(* Logix 5000 project; controller GEA_Test_Chamber vendor 1 type 14 code 196 rev 32.14; software revision 32.04; part 5 of 11 *)
(* tags used below, declared in another part *)
   Wrk_Index : DINT;
(* raC_Tec_NetModbusTCPServer_RespStrWord, continued *)

ROUTINE Prescan   (* ladder *)
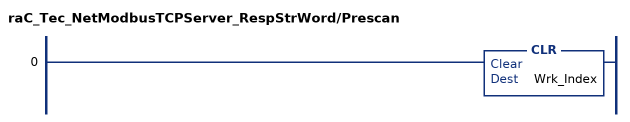
   0: CLR(Wrk_Index);
END_ROUTINE
END_ADD_ON_INSTRUCTION

ADD_ON_INSTRUCTION T_DIFF   (* revision 1.0 *)
VAR_IN_OUT
   TimeRef : DINT[7]; {required}
   ActTime : DINT[7]; {required}
END_VAR
VAR_OUTPUT
   T_Diff_sec : DINT; {required}
END_VAR
VAR
   Temp_Time : DINT[7]; {access None}
   sec : DINT[3]; {access None}
END_VAR

ROUTINE Logic   (* ladder *)
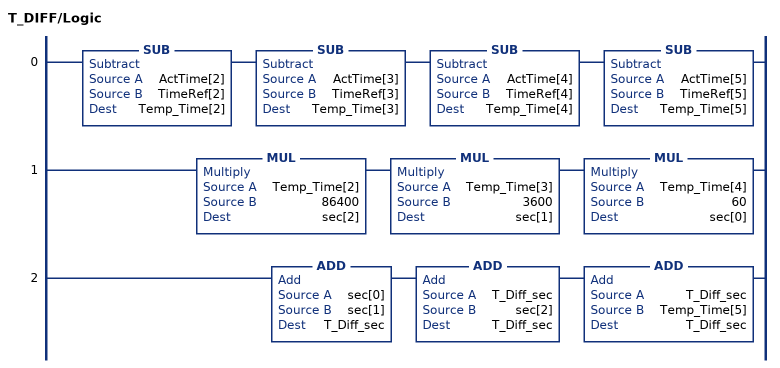
   0: SUB(ActTime[2],TimeRef[2],Temp_Time[2])SUB(ActTime[3],TimeRef[3],Temp_Time[3])SUB(ActTime[4],TimeRef[4],Temp_Time[4])SUB(ActTime[5],TimeRef[5],Temp_Time[5]);
   1: MUL(Temp_Time[2],86400,sec[2])MUL(Temp_Time[3],3600,sec[1])MUL(Temp_Time[4],60,sec[0]);
   2: ADD(sec[0],sec[1],T_Diff_sec)ADD(T_Diff_sec,sec[2],T_Diff_sec)ADD(T_Diff_sec,Temp_Time[5],T_Diff_sec);
END_ROUTINE
END_ADD_ON_INSTRUCTION

VAR_GLOBAL   (* controller tags *)
   always_off : BOOL;
   Amount_Water_Flow : DINT := 200;
   Client_01 : raC_Opr_NetModbusTCPClient := (Inp_Enable := 1, Sts_EN := 1, Sts_Connected := 1);
   Client_01_Data : raC_UDT_ModbusClientData := (Coils_0xxx[0] := 1, Coils_0xxx[1] := 1, Coils_0xxx[2] := 1, Coils_0xxx[3] := 1, Coils_0xxx[1010] := 1, Coils_0xxx[1012] := 1, Coils_0xxx[1014] := 1, Coils_0xxx[1015] := 1, HoldRegisters_4xxx[0] := 10, HoldRegisters_4xxx[1] := 512, HoldRegisters_4xxx[32] := 102, HoldRegisters_4xxx[33] := 2330);
   Client_01_EN : BOOL := 1;
   Client_01_MSG_Connect : MESSAGE;
        MessageParameters(ServiceCode := 16#004c, LocalElement := Client_01_Parameters.MSG_Src[0], ...)
   Client_01_MSG_Create : MESSAGE;
        MessageParameters(ServiceCode := 16#004b, LocalElement := Client_01_Parameters.MSG_Src[0], DestinationTag := Client_01_Parameters.MSG_Dest[0], ...)
   Client_01_MSG_Delete : MESSAGE;
        MessageParameters(ServiceCode := 16#004f, ...)
   Client_01_MSG_Read : MESSAGE;
        MessageParameters(ServiceCode := 16#004d, LocalElement := Client_01_Parameters.MSG_Src[0], DestinationTag := Client_01_Parameters.MSG_Dest[0], ...)
   Client_01_MSG_SetSing : MESSAGE;
        MessageParameters(ServiceCode := 16#0010, LocalElement := Client_01_Parameters.MSG_Src[496], ...)
   Client_01_MSG_Write : MESSAGE;
        MessageParameters(ServiceCode := 16#004e, LocalElement := Client_01_Parameters.MSG_Src[0], DestinationTag := Client_01_Parameters.MSG_Dest[0], ...)
   Client_01_Parameters : raC_UDT_ModbusClientConnection := (DestAddress := '10.2.0.15', DestinationPort := 502, MSG_Src[4] := -28, MSG_Src[5] := 1, MSG_Src[12] := 12, MSG_Src[16] := 58, MSG_Src[17] := 106, MSG_Src[21] := 6, MSG_Src[22] := 1, MSG_Src[23] := 4, MSG_Src[25] := 3, MSG_Src[27] := 10, MSG_Src[28] := 50, MSG_Src[29] := 50, MSG_Src[496] := 1, MSG_Dest[12] := 58, MSG_Dest[13] := 105, MSG_Dest[17] := 23, MSG_Dest[18] := 1, MSG_Dest[19] := 4, MSG_Dest[20] := 20, MSG_Dest[86] := 102, MSG_Dest[87] := 9, MSG_Dest[88] := 26, MSG_Dest[232] := 105, MSG_Dest[233] := 29, MSG_Dest[237] := 6, MSG_Dest[239] := 6);
   Client_01_Transactions : raC_UDT_ModbusClientTransaction[5] := ([0].Enabled := 1, [0].PollInterval := 500, [0].TransType := 4, [0].StationID := 1, [0].BeginAddress := 3, [0].Count := 10, [0].TransComplete := 1, [0].Diagnostic.Request := ':h$00$00$00$06$01$04$00$03$00$0A', [0].Diagnostic.TransID := 14952, [0].Diagnostic.IntervalTimer.PRE := 460, [0].Diagnostic.IntervalTimer.ACC := 395, [0].Diagnostic.IntervalTimer.EN := 1, [0].Diagnostic.IntervalTimer.TT := 1, [0].Diagnostic.NoReplyCounter.PRE := 10, [0].Diagnostic.PendingTimer.PRE := 3000, [1].PollInterval := 1000, [1].Diagnostic.IntervalTimer.PRE := 960, [1].Diagnostic.IntervalTimer.ACC := 960, [1].Diagnostic.IntervalTimer.EN := 1, [1].Diagnostic.IntervalTimer.DN := 1, [1].Diagnostic.NoReplyCounter.PRE := 10, [1].Diagnostic.PendingTimer.PRE := 3000, [2].PollInterval := 1000, [2].Diagnostic.IntervalTimer.PRE := 960, [2].Diagnostic.IntervalTimer.ACC := 960, [2].Diagnostic.IntervalTimer.EN := 1, [2].Diagnostic.IntervalTimer.DN := 1, [2].Diagnostic.NoReplyCounter.PRE := 10, [2].Diagnostic.PendingTimer.PRE := 3000, [3].PollInterval := 1000, [3].Diagnostic.IntervalTimer.PRE := 960, [3].Diagnostic.IntervalTimer.ACC := 960, [3].Diagnostic.IntervalTimer.EN := 1, [3].Diagnostic.IntervalTimer.DN := 1, [3].Diagnostic.NoReplyCounter.PRE := 10, [3].Diagnostic.PendingTimer.PRE := 3000, [4].PollInterval := 1000, [4].Diagnostic.IntervalTimer.PRE := 960, [4].Diagnostic.IntervalTimer.ACC := 369, [4].Diagnostic.IntervalTimer.EN := 1, [4].Diagnostic.IntervalTimer.DN := 1, [4].Diagnostic.NoReplyCounter.PRE := 10, [4].Diagnostic.PendingTimer.PRE := 3000);
   Client_02 : raC_Opr_NetModbusTCPClient := (Inp_Enable := 1, Sts_EN := 1, Sts_Connected := 1);
   Client_02_Data : raC_UDT_ModbusClientData := (Coils_0xxx[0] := 1, Coils_0xxx[1] := 1, Coils_0xxx[2] := 1, Coils_0xxx[3] := 1, Coils_0xxx[1010] := 1, Coils_0xxx[1012] := 1, Coils_0xxx[1014] := 1, Coils_0xxx[1015] := 1, InpRegisters_3xxx[3] := 159, InpRegisters_3xxx[7] := 1904);
   Client_02_EN : BOOL := 1;
   Client_02_MSG_Connect : MESSAGE;
        MessageParameters(ServiceCode := 16#004c, LocalElement := Client_02_Parameters.MSG_Src[0], ...)
   Client_02_MSG_Create : MESSAGE;
        MessageParameters(ServiceCode := 16#004b, LocalElement := Client_02_Parameters.MSG_Src[0], DestinationTag := Client_02_Parameters.MSG_Dest[0], ...)
   Client_02_MSG_Delete : MESSAGE;
        MessageParameters(ServiceCode := 16#004f, ...)
   Client_02_MSG_Read : MESSAGE;
        MessageParameters(ServiceCode := 16#004d, LocalElement := Client_02_Parameters.MSG_Src[0], DestinationTag := Client_02_Parameters.MSG_Dest[0], ...)
   Client_02_MSG_SetSing : MESSAGE;
        MessageParameters(ServiceCode := 16#0010, LocalElement := Client_02_Parameters.MSG_Src[496], ...)
   Client_02_MSG_Write : MESSAGE;
        MessageParameters(ServiceCode := 16#004e, LocalElement := Client_02_Parameters.MSG_Src[0], DestinationTag := Client_02_Parameters.MSG_Dest[0], ...)
   Client_02_Parameters : raC_UDT_ModbusClientConnection := (DestAddress := '10.2.0.14', DestinationPort := 502, MSG_Src[4] := -28, MSG_Src[5] := 1, MSG_Src[12] := 12, MSG_Src[16] := 63, MSG_Src[17] := 53, MSG_Src[21] := 6, MSG_Src[22] := 1, MSG_Src[23] := 4, MSG_Src[25] := 3, MSG_Src[27] := 10, MSG_Src[28] := 20, MSG_Src[496] := 1, MSG_Dest[12] := 63, MSG_Dest[13] := 52, MSG_Dest[17] := 23, MSG_Dest[18] := 1, MSG_Dest[19] := 4, MSG_Dest[20] := 20, MSG_Dest[28] := -97, MSG_Dest[35] := 7, MSG_Dest[36] := 112, MSG_Dest[42] := 1, MSG_Dest[43] := -122, MSG_Dest[44] := -96, MSG_Dest[45] := 48, MSG_Dest[46] := 50, MSG_Dest[47] := 48, MSG_Dest[48] := 46, MSG_Dest[49] := 51, MSG_Dest[50] := 52, MSG_Dest[51] := 32, MSG_Dest[52] := 48, MSG_Dest[53] := 48, MSG_Dest[54] := 50, MSG_Dest[55] := 48, MSG_Dest[56] := 46, MSG_Dest[57] := 51, MSG_Dest[58] := 52, MSG_Dest[59] := 32, MSG_Dest[60] := 48, MSG_Dest[61] := 48, MSG_Dest[62] := 50, MSG_Dest[63] := 48, MSG_Dest[64] := 46, MSG_Dest[65] := 51, MSG_Dest[66] := 52, MSG_Dest[67] := 32, MSG_Dest[68] := 48, MSG_Dest[69] := 48, MSG_Dest[70] := 50, MSG_Dest[71] := 48, MSG_Dest[72] := 46, MSG_Dest[73] := 51, MSG_Dest[74] := 52, MSG_Dest[75] := 32, MSG_Dest[76] := 48, MSG_Dest[77] := 48, MSG_Dest[78] := 50,
        MSG_Dest[79] := 48, MSG_Dest[80] := 46, MSG_Dest[81] := 51, MSG_Dest[82] := 52, MSG_Dest[83] := 32, MSG_Dest[84] := 48, MSG_Dest[85] := 48, MSG_Dest[86] := 50, MSG_Dest[87] := 48, MSG_Dest[88] := 46, MSG_Dest[89] := 51, MSG_Dest[90] := 52, MSG_Dest[91] := 32, MSG_Dest[92] := 48, MSG_Dest[93] := 48, MSG_Dest[94] := 50, MSG_Dest[95] := 48, MSG_Dest[96] := 46, MSG_Dest[97] := 51, MSG_Dest[98] := 52, MSG_Dest[99] := 32, MSG_Dest[100] := 48, MSG_Dest[101] := 48, MSG_Dest[102] := 50, MSG_Dest[103] := 48, MSG_Dest[104] := 46, MSG_Dest[105] := 51, MSG_Dest[106] := 52, MSG_Dest[107] := 32, MSG_Dest[108] := 48, MSG_Dest[109] := 48, MSG_Dest[110] := 50, MSG_Dest[111] := 48, MSG_Dest[112] := 46, MSG_Dest[113] := 51, MSG_Dest[114] := 52, MSG_Dest[115] := 32, MSG_Dest[116] := 48, MSG_Dest[117] := 48, MSG_Dest[118] := 50, MSG_Dest[119] := 48, MSG_Dest[120] := 46, MSG_Dest[121] := 51, MSG_Dest[122] := 52, MSG_Dest[123] := 32, MSG_Dest[124] := 48, MSG_Dest[125] := 48, MSG_Dest[126] := 50, MSG_Dest[127] := 48, MSG_Dest[128] := 46, MSG_Dest[129] := 51, MSG_Dest[130] := 52, MSG_Dest[131] := 32, MSG_Dest[132] := 48, MSG_Dest[133] := 48, MSG_Dest[134] := 50, MSG_Dest[135] := 48, MSG_Dest[136] := 46, MSG_Dest[137] := 51, MSG_Dest[138] := 52,
        MSG_Dest[139] := 32, MSG_Dest[140] := 48, MSG_Dest[141] := 48, MSG_Dest[142] := 50, MSG_Dest[143] := 48, MSG_Dest[144] := 46, MSG_Dest[145] := 51, MSG_Dest[146] := 52, MSG_Dest[147] := 32, MSG_Dest[148] := 48, MSG_Dest[149] := 48, MSG_Dest[150] := 50, MSG_Dest[151] := 48, MSG_Dest[152] := 46, MSG_Dest[153] := 51, MSG_Dest[154] := 52, MSG_Dest[155] := 32, MSG_Dest[156] := 48, MSG_Dest[157] := 48, MSG_Dest[158] := 50, MSG_Dest[159] := 48, MSG_Dest[160] := 46, MSG_Dest[161] := 51, MSG_Dest[162] := 52, MSG_Dest[163] := 32, MSG_Dest[164] := 48, MSG_Dest[165] := 48, MSG_Dest[166] := 50, MSG_Dest[167] := 48, MSG_Dest[168] := 46, MSG_Dest[169] := 51, MSG_Dest[170] := 52, MSG_Dest[171] := 32, MSG_Dest[172] := 48, MSG_Dest[173] := 48, MSG_Dest[174] := 50, MSG_Dest[175] := 48, MSG_Dest[176] := 46, MSG_Dest[177] := 51, MSG_Dest[178] := 52, MSG_Dest[179] := 32, MSG_Dest[180] := 48, MSG_Dest[181] := 48, MSG_Dest[182] := 50, MSG_Dest[183] := 48, MSG_Dest[184] := 46, MSG_Dest[185] := 51, MSG_Dest[186] := 52, MSG_Dest[187] := 32, MSG_Dest[188] := 48, MSG_Dest[189] := 48, MSG_Dest[190] := 50, MSG_Dest[191] := 48, MSG_Dest[192] := 46, MSG_Dest[193] := 51, MSG_Dest[194] := 52, MSG_Dest[195] := 32, MSG_Dest[196] := 48, MSG_Dest[197] := 48, MSG_Dest[198] := 50,
        MSG_Dest[199] := 48, MSG_Dest[200] := 46, MSG_Dest[201] := 51, MSG_Dest[202] := 52, MSG_Dest[203] := 32, MSG_Dest[204] := 48, MSG_Dest[205] := 48, MSG_Dest[206] := 50, MSG_Dest[207] := 48, MSG_Dest[208] := 46, MSG_Dest[209] := 51, MSG_Dest[210] := 52, MSG_Dest[211] := 32, MSG_Dest[212] := 48, MSG_Dest[213] := 48, MSG_Dest[214] := 50, MSG_Dest[215] := 48, MSG_Dest[216] := 46, MSG_Dest[217] := 51, MSG_Dest[218] := 52, MSG_Dest[219] := 32, MSG_Dest[220] := 48, MSG_Dest[221] := 48, MSG_Dest[222] := 50, MSG_Dest[223] := 48, MSG_Dest[224] := 46, MSG_Dest[225] := 51, MSG_Dest[226] := 52, MSG_Dest[227] := 32, MSG_Dest[228] := 48, MSG_Dest[229] := 48, MSG_Dest[230] := 50, MSG_Dest[231] := 48, MSG_Dest[232] := 46, MSG_Dest[233] := 51, MSG_Dest[234] := 52, MSG_Dest[235] := 32, MSG_Dest[236] := 48, MSG_Dest[237] := 48, MSG_Dest[238] := 50, MSG_Dest[239] := 48, MSG_Dest[240] := 46, MSG_Dest[241] := 51, MSG_Dest[242] := 52, MSG_Dest[243] := 32, MSG_Dest[244] := 48, MSG_Dest[245] := 48, MSG_Dest[246] := 50, MSG_Dest[247] := 48, MSG_Dest[248] := 46, MSG_Dest[249] := 51, MSG_Dest[250] := 52, MSG_Dest[251] := 32, MSG_Dest[252] := 48, MSG_Dest[253] := 48, MSG_Dest[254] := 50, MSG_Dest[255] := 48, MSG_Dest[256] := 46, MSG_Dest[257] := 51, MSG_Dest[258] := 52,
        MSG_Dest[259] := 32, MSG_Dest[260] := 48, MSG_Dest[261] := 48, MSG_Dest[262] := 50, MSG_Dest[263] := 48, MSG_Dest[264] := 46, MSG_Dest[265] := 51, MSG_Dest[266] := 52, MSG_Dest[267] := 32);
   Client_02_Transactions : raC_UDT_ModbusClientTransaction[5] := ([0].Enabled := 1, [0].PollInterval := 500, [0].TransType := 4, [0].StationID := 1, [0].BeginAddress := 3, [0].Count := 10, [0].TransStat := 1, [0].Diagnostic.Request := '?4$00$00$00$06$01$04$00$03$00$0A', [0].Diagnostic.ReqBuilt := 1, [0].Diagnostic.TransID := 16180, [0].Diagnostic.IntervalTimer.PRE := 460, [0].Diagnostic.IntervalTimer.ACC := 44, [0].Diagnostic.IntervalTimer.EN := 1, [0].Diagnostic.IntervalTimer.TT := 1, [0].Diagnostic.NoReplyCounter.PRE := 10, [0].Diagnostic.PendingTimer.PRE := 3000, [0].Diagnostic.PendingTimer.ACC := 44, [0].Diagnostic.PendingTimer.EN := 1, [0].Diagnostic.PendingTimer.TT := 1, [1].PollInterval := 1000, [1].Diagnostic.IntervalTimer.PRE := 960, [1].Diagnostic.IntervalTimer.ACC := 960, [1].Diagnostic.IntervalTimer.EN := 1, [1].Diagnostic.IntervalTimer.DN := 1, [1].Diagnostic.NoReplyCounter.PRE := 10, [1].Diagnostic.PendingTimer.PRE := 3000, [2].PollInterval := 1000, [2].Diagnostic.IntervalTimer.PRE := 960, [2].Diagnostic.IntervalTimer.ACC := 960, [2].Diagnostic.IntervalTimer.EN := 1, [2].Diagnostic.IntervalTimer.DN := 1, [2].Diagnostic.NoReplyCounter.PRE := 10, [2].Diagnostic.PendingTimer.PRE := 3000, [3].PollInterval := 1000, [3].Diagnostic.IntervalTimer.PRE := 960, [3].Diagnostic.IntervalTimer.ACC := 369, [3].Diagnostic.IntervalTimer.EN := 1, [3].Diagnostic.IntervalTimer.DN := 1, [3].Diagnostic.NoReplyCounter.PRE := 10, [3].Diagnostic.PendingTimer.PRE := 3000, [4].PollInterval := 1000, [4].Diagnostic.IntervalTimer.PRE := 960, [4].Diagnostic.IntervalTimer.ACC := 369, [4].Diagnostic.IntervalTimer.EN := 1, [4].Diagnostic.IntervalTimer.DN := 1, [4].Diagnostic.NoReplyCounter.PRE := 10, [4].Diagnostic.PendingTimer.PRE := 3000);
   Control_Off : BOOL;
   FVIR_Error_MSG : INT := 131;
   FVIR_LabView_Control : INT := 33;
        .1   // 1 - Start Test / 0 - Stop Test
        .3   // Water Outlet Valve, 1 - Open, 0 - Close
        .4   // Water Intlet Valve, 1 - Open, 0 - Close
        .5   // Gas Solenoid Valve, 1 - Open, 0 - Close
        .2   // Start Mannequin Sequence (When test is stopped)
        .11   // Actruator Spill Gasoline Go To Home Pos
        .12   // Actruator Spill Gasoline Go To Work Pos
        .0   // Life Bit
        .13   // Reset Laurel Flow Meter
        .10   // Actruator Mannequin Go To Work Pos
        .9   // Actruator Mannequin Go To Home Pos
        .7   // Reserve
        .6   // Water Flow Intellifaucet DRK375, 1 - Start puls (1 sec)
        .8   // Water Flow Intellifaucet DRK375, 1 - Stop puls (1 sec)
        .15   // Water Outlet Proportional Valve 0 - PID controls the Flow, 1 - PID controls the Temperature
        .14   // Water Heater Status, 1 - Burner ON, 0 - Standby
   FVIR_LabView_Status : INT := 288;
        .2   // Spill Gasoline Can in Progress
        .1   // Mannequin Movement Sequence in Progress
        .3   // Water Outlet Valve, 1 - Open, 0 - Close
        .4   // Water Intlet Valve, 1 - Open, 0 - Close
        .5   // Gas Solenoid Valve, 1 - Open, 0 - Close
        .10   // Actruator Spill Gasoline Go To Home Pos
        .11   // Actruator Spill Gasoline Go To Work Pos
        .0   // Life Bit
        .6   // Water Flow Intellifaucet DRK375, 1 - Open, 0 - Close
        .8   // Actruator Mannequin Go To Home Pos
        .7   // 1 - Test Chamber In Sequence/0 - Test is stopped
        .14   // Spare
        .15   // Reset FVIR Totalizer
        .9   // Actruator Mannequin Go To Work Pos
        .12   // 1 - Start recording data
        .13   // Water Outlet Flow Proportional Valve EPV-312B 1 - Open, 0 - Close
   FVIR_Mannequin_Direction_TimeDelay : INT := 1300;
   FVIR_Mannequin_Time_Pause : INT := 60;
   FVIR_Number_Mannequin_Movement : INT := 3;
   FVIR_Rate_REAL : REAL;
   FVIR_Reset_Cnt : BOOL;
   FVIR_Reset_Cnt_inprogress : BOOL;
   FVIR_Test_No : INT;
   FVIR_Totalizer_REAL : REAL;
   FVIR_Water_Flow_DRK375 : INT := 15;
   FVIR_Water_Flow_DRK375_Float : REAL := 100.0;
   FVIR_Water_Outlet_Valve : INT := 3;
   FVIR_Water_Outlet_Valve_Flow_SP : REAL;
   FVIR_Water_Outlet_Valve_SP : REAL := 3.0;
   FVIR_Water_Temp_DRK375 : INT := 70;
   FVIR_Water_Temp_DRK375_Float : REAL := 70.0;
   Heater_Cnt : COUNTER := (ACC := 121, DN := 1);
   LDO_BurnerCycle_11_12_OFF : INT := 5;
   LDO_BurnerCycle_11_12_ON : INT := 235;
   LDO_BurnerCycle_13_OFF : INT := 5;
   LDO_BurnerCycle_13_ON : INT := 55;
   LDO_BurnerCycle_1_10_OFF : INT := 5;
   LDO_BurnerCycle_1_10_ON : INT := 55;
   LDO_Error_MSG : INT := 126;
   LDO_LabView_Control : INT := 24612;
        .3   // Water Outlet Valve, 1 - Open, 0 - Close
        .4   // Water Intlet Valve, 1 - Open, 0 - Close
        .5   // Gas Solenoid Valve, 1 - Open, 0 - Close
        .2   // 1 - Start Test / 0 - Stop Test
        .1   // Spare
        .0   // Life Bit
        .10   // Oil spray 1.1cc/min
        .6   // Water Flow Intellifaucet DRK375, Start
        .13   // Reset Laurel Flow Meter
        .11   // Oil spray 1.33cc/min
        .9   // Oil spray 0.8cc/min
        .12   // Heater ON/0 - Heater OFF
        .7   // Water Outlet Flow Proportional Valve EPV-312B 1 - Open, 0 - Close
        .8   // Water Flow Intellifaucet DRK375, Stop
        .14   // Burner ON
        .15   // PID selector, 1 - Temperature control, 0 - Flow control
   LDO_LabView_Control2 : INT;
        .0   // Conveyors Turn On
        .7   // Blower Turn On
   LDO_LabView_Status : INT := 2080;
        .3   // Water Outlet Valve, 1 - Open, 0 - Close
        .4   // Water Intlet Valve, 1 - Open, 0 - Close
        .5   // Gas Solenoid Valve, 1 - Open, 0 - Close
        .11   // Heater ON/OFF, 1 - ON, 0 - OFF
        .8   // Oil spray 0.8cc/min, 1 - Open, 0 - Close
        .7   // 1 - Test Chamber In Sequence/0 - Test is stopped
        .2   // Spare
        .12   // Spare
        .0   // Life Bit
        .6   // Water Flow Intellifaucet DRK375, 1 - Open, 0 - Close
        .1   // Start recording data
        .10   // Oil spray 1.33cc/min, 1 - Open, 0 - Close
        .13   // Spare
        .14   // Spare
        .15   // Spare
        .9   // Oil spray 1.1cc/min, 1 - Open, 0 - Close
   LDO_Oil_1st_seq_OFF : INT := 25;
   LDO_Oil_1st_seq_ON : INT := 5;
   LDO_Oil_all_seq_OFF : INT := 27;
   LDO_Oil_all_seq_ON : INT := 3;
   LDO_Oil_pre_seq_OFF : INT := 20;
   LDO_Oil_pre_seq_ON : INT := 10;
   LDO_Reset_Cnt : BOOL;
   LDO_Reset_CNT_inprogress : BOOL;
   LDO_Water_Flow_DRK375 : INT := 96;
   LDO_Water_Flow_DRK375_Float : REAL := 50.0;
   LDO_Water_Outlet_Valve : REAL;
   LDO_Water_Outlet_Valve_Flow_SP : REAL := 0.5803782;
   LDO_Water_Outlet_Valve_SP : REAL := 135.0;
   LDO_Water_Temp_DRK375 : INT := 32;
   LDO_Water_Temp_DRK375_Float : REAL := 70.0;
   Marcin : BOOL;
   Modbus_LabView : raC_Opr_NetModbusTCPServer := (Inp_Enable := 1, Sts_EN := 1, Sts_Waiting := 1, Sts_LastError := -4);
   Modbus_LabView_Data : raC_UDT_ModbusServerData := (Coils_0xxx[1] := 1, Coils_0xxx[2] := 1, InpRegisters_3xxx[0] := 288, InpRegisters_3xxx[1] := 131, InpRegisters_3xxx[2] := 695, InpRegisters_3xxx[3] := 689, InpRegisters_3xxx[4] := 688, InpRegisters_3xxx[5] := 698, InpRegisters_3xxx[6] := 898, InpRegisters_3xxx[7] := 859, InpRegisters_3xxx[8] := 678, InpRegisters_3xxx[9] := -1495, InpRegisters_3xxx[10] := 671, InpRegisters_3xxx[11] := 1181, InpRegisters_3xxx[12] := -3497, InpRegisters_3xxx[13] := -3470, InpRegisters_3xxx[14] := -3508, InpRegisters_3xxx[15] := -3483, InpRegisters_3xxx[16] := -3499, InpRegisters_3xxx[17] := -3480, InpRegisters_3xxx[18] := -3290, InpRegisters_3xxx[19] := -3270, InpRegisters_3xxx[20] := -3280, InpRegisters_3xxx[21] := -3275, InpRegisters_3xxx[22] := 684, InpRegisters_3xxx[23] := 687, InpRegisters_3xxx[24] := 690, InpRegisters_3xxx[25] := 681, InpRegisters_3xxx[26] := 1000, InpRegisters_3xxx[28] := -50, InpRegisters_3xxx[29] := -50, InpRegisters_3xxx[31] := 2080, InpRegisters_3xxx[32] := 126, InpRegisters_3xxx[33] := 1006, InpRegisters_3xxx[34] := 956, InpRegisters_3xxx[35] := 732, InpRegisters_3xxx[36] := 776, InpRegisters_3xxx[37] := 728, InpRegisters_3xxx[38] := 728, InpRegisters_3xxx[39] := 724, InpRegisters_3xxx[40] := 721, InpRegisters_3xxx[41] := 741, InpRegisters_3xxx[42] := 746, InpRegisters_3xxx[43] := 1355, InpRegisters_3xxx[44] := 21870, InpRegisters_3xxx[45] := 21870, InpRegisters_3xxx[46] := 21870, InpRegisters_3xxx[47] := 24966, InpRegisters_3xxx[48] := 24966, InpRegisters_3xxx[49] := 24966, InpRegisters_3xxx[50] := 24966, InpRegisters_3xxx[51] := 4270, InpRegisters_3xxx[52] := 2540, InpRegisters_3xxx[53] := 40, InpRegisters_3xxx[57] := 26214, InpRegisters_3xxx[58] := 17214, InpRegisters_3xxx[59] := 1, InpRegisters_3xxx[60] := 1, InpRegisters_3xxx[61] := 14, InpRegisters_3xxx[62] := 121,
        InpRegisters_3xxx[63] := 2022, InpRegisters_3xxx[64] := 8, InpRegisters_3xxx[65] := 30, InpRegisters_3xxx[67] := 36, InpRegisters_3xxx[68] := 14, InpRegisters_3xxx[69] := 2, InpRegisters_3xxx[71] := 22, InpRegisters_3xxx[73] := 48, HoldRegisters_4xxx[0] := 33, HoldRegisters_4xxx[1] := 1300, HoldRegisters_4xxx[2] := 3, HoldRegisters_4xxx[3] := 3, HoldRegisters_4xxx[4] := 70, HoldRegisters_4xxx[5] := 15, HoldRegisters_4xxx[6] := 60, HoldRegisters_4xxx[10] := 24612, HoldRegisters_4xxx[14] := 17036, HoldRegisters_4xxx[16] := 16968, HoldRegisters_4xxx[18] := 17159, HoldRegisters_4xxx[19] := 55, HoldRegisters_4xxx[20] := 5, HoldRegisters_4xxx[21] := 235, HoldRegisters_4xxx[22] := 5, HoldRegisters_4xxx[23] := 55, HoldRegisters_4xxx[24] := 5, HoldRegisters_4xxx[25] := 5, HoldRegisters_4xxx[26] := 25, HoldRegisters_4xxx[27] := 3, HoldRegisters_4xxx[28] := 27, HoldRegisters_4xxx[29] := 10, HoldRegisters_4xxx[30] := 20, HoldRegisters_4xxx[31] := -27734, HoldRegisters_4xxx[32] := 16148, HoldRegisters_4xxx[34] := 200, HoldRegisters_4xxx[52] := 17036, HoldRegisters_4xxx[54] := 17096, HoldRegisters_4xxx[56] := 16448);
   Modbus_LabView_EN : BOOL := 1;
   Modbus_LabView_MSG_Accept : MESSAGE;
        MessageParameters(ServiceCode := 16#0050, LocalElement := Modbus_LabView_Parameters.MSG_Src[500], DestinationTag := Modbus_LabView_Parameters.MSG_Dest[500], ...)
   Modbus_LabView_MSG_Create : MESSAGE;
        MessageParameters(ServiceCode := 16#004b, LocalElement := Modbus_LabView_Parameters.MSG_Src[0], DestinationTag := Modbus_LabView_Parameters.MSG_Dest[0], ...)
   Modbus_LabView_MSG_Delete : MESSAGE;
        MessageParameters(ServiceCode := 16#004f, ...)
   Modbus_LabView_MSG_DeleteAll : MESSAGE;
        MessageParameters(ServiceCode := 16#0051, ...)
   Modbus_LabView_MSG_Read : MESSAGE;
        MessageParameters(ServiceCode := 16#004d, LocalElement := Modbus_LabView_Parameters.MSG_Src[0], DestinationTag := Modbus_LabView_Parameters.MSG_Dest[0], ...)
   Modbus_LabView_MSG_SetSing : MESSAGE;
        MessageParameters(ServiceCode := 16#0010, LocalElement := Modbus_LabView_Parameters.MSG_Src[496], ...)
   Modbus_LabView_MSG_Write : MESSAGE;
        MessageParameters(ServiceCode := 16#004e, LocalElement := Modbus_LabView_Parameters.MSG_Src[0], DestinationTag := Modbus_LabView_Parameters.MSG_Dest[0], ...)
   Modbus_LabView_Parameters : raC_UDT_ModbusServerBase := (LocalPort := 502, InactivityTimeout := 60, MSG_Src[4] := -28, MSG_Src[5] := 1, MSG_Src[12] := 17, MSG_Src[16] := 50, MSG_Src[17] := -72, MSG_Src[21] := 11, MSG_Src[22] := 1, MSG_Src[23] := 4, MSG_Src[24] := 8, MSG_Src[33] := 2, MSG_Src[34] := -77, MSG_Src[35] := 2, MSG_Src[36] := -67, MSG_Src[37] := 3, MSG_Src[38] := -98, MSG_Src[39] := 3, MSG_Src[40] := 103, MSG_Src[41] := 2, MSG_Src[42] := -86, MSG_Src[43] := -6, MSG_Src[44] := 41, MSG_Src[45] := 2, MSG_Src[46] := -86, MSG_Src[47] := 4, MSG_Src[48] := -83, MSG_Src[49] := -14, MSG_Src[50] := 87, MSG_Src[51] := -14, MSG_Src[52] := 114, MSG_Src[53] := -14, MSG_Src[54] := 76, MSG_Src[55] := -14, MSG_Src[56] := 101, MSG_Src[57] := -14, MSG_Src[58] := 85, MSG_Src[59] := -14, MSG_Src[60] := 104, MSG_Src[61] := -13, MSG_Src[62] := 38, MSG_Src[63] := -13, MSG_Src[64] := 58, MSG_Src[65] := -13, MSG_Src[66] := 48, MSG_Src[67] := -13, MSG_Src[68] := 53, MSG_Src[69] := 2, MSG_Src[70] := -85, MSG_Src[71] := 2, MSG_Src[72] := -82, MSG_Src[73] := 2, MSG_Src[74] := -87, MSG_Src[75] := 2, MSG_Src[76] := -77, MSG_Src[77] := 3, MSG_Src[78] := -24, MSG_Src[81] := -1, MSG_Src[82] := -50, MSG_Src[83] := -1,
        MSG_Src[84] := -50, MSG_Src[87] := 120, MSG_Src[88] := -5, MSG_Src[90] := 122, MSG_Src[91] := 2, MSG_Src[92] := -68, MSG_Src[93] := 4, MSG_Src[94] := -77, MSG_Src[95] := 2, MSG_Src[96] := -19, MSG_Src[97] := 3, MSG_Src[98] := -83, MSG_Src[99] := 2, MSG_Src[100] := 48, MSG_Src[101] := 3, MSG_Src[102] := 12, MSG_Src[103] := 2, MSG_Src[104] := -69, MSG_Src[105] := 2, MSG_Src[106] := -44, MSG_Src[107] := 3, MSG_Src[108] := 15, MSG_Src[109] := 2, MSG_Src[110] := -19, MSG_Src[111] := 8, MSG_Src[112] := -92, MSG_Src[113] := 85, MSG_Src[114] := 110, MSG_Src[115] := 85, MSG_Src[116] := 110, MSG_Src[117] := 85, MSG_Src[118] := 110, MSG_Src[119] := 97, MSG_Src[120] := -122, MSG_Src[121] := 97, MSG_Src[122] := -122, MSG_Src[123] := 97, MSG_Src[124] := -122, MSG_Src[125] := 97, MSG_Src[126] := -122, MSG_Src[127] := 7, MSG_Src[128] := -68, MSG_Src[129] := 9, MSG_Src[130] := -40, MSG_Src[131] := 5, MSG_Src[132] := 90, MSG_Src[133] := 10, MSG_Src[134] := -56, MSG_Src[135] := 81, MSG_Src[136] := -20, MSG_Src[137] := 62, MSG_Src[138] := -72, MSG_Src[139] := 76, MSG_Src[140] := -51, MSG_Src[141] := 67, MSG_Src[142] := 62, MSG_Src[144] := 1, MSG_Src[146] := 1, MSG_Src[148] := 14, MSG_Src[150] := 12,
        MSG_Src[151] := 7, MSG_Src[152] := -26, MSG_Src[154] := 8, MSG_Src[156] := 25, MSG_Src[158] := 8, MSG_Src[160] := 53, MSG_Src[162] := 31, MSG_Src[496] := 1, MSG_Src[500] := 10, MSG_Dest[12] := 50, MSG_Dest[13] := -72, MSG_Dest[17] := 6, MSG_Dest[18] := 1, MSG_Dest[19] := 4, MSG_Dest[21] := 79, MSG_Dest[23] := 4, MSG_Dest[24] := 4, MSG_Dest[25] := -109, MSG_Dest[26] := -86, MSG_Dest[27] := 63, MSG_Dest[28] := 20, MSG_Dest[38] := 100, MSG_Dest[39] := -13, MSG_Dest[40] := 66, MSG_Dest[41] := -46, MSG_Dest[500] := -126, MSG_Dest[501] := 72, MSG_Dest[504] := 2, MSG_Dest[506] := 79, MSG_Dest[507] := -39, MSG_Dest[508] := 8, MSG_Dest[510] := 2, MSG_Dest[511] := 10);
   nLDO_Rate_REAL : REAL;
   nLDO_Totalizer_REAL : REAL := 190.4;
   Oil_inj_08_Cnt : COUNTER := (ACC := 1, DN := 1);
   Oil_inj_11_Cnt : COUNTER := (ACC := 1, DN := 1);
   Oil_inj_133_Cnt : COUNTER := (ACC := 14, DN := 1);
   Output_FVIR : Output_FVIR := (Actuation_Mannequin_Base := 1, Gas_Solenoid_Valve := 1, Water_Temperature_Flow_Control := 3093);
   Output_LDO : Output_LDO := (Gas_Solenoid_Valve := 1, Water_Temperature_Flow_Control := 3093);
   pulsReset : BOOL;
   SET_0 : BOOL;
   SET_1 : BOOL := 1;
   Timer_Delay_Start : TIMER := (PRE := 200000);
   TimeUTC : DINT[6] := ([0] := 2021663793, [1] := 207765);
   Water_Flow_DRK375_Last_Float : REAL := 50.0;
END_VAR

PROGRAM FVIR_Chamber   (* main routine FVIR_Main *)
VAR
   bPulse05Hz : BOOL := 1;
   bPulse0_1Hz : BOOL := 1;
   bPulse10Hz : BOOL;
   bPulse1Hz : BOOL;
   Cycle_Counter : SINT;
   DRK375_Flow_Change : BOOL;
   DRK375_Flow_InRange : BOOL := 1;
   DRK375_Temp_Change : BOOL;
   DRK375_Temp_InRange : BOOL := 1;
   Error_MSG : INT := 131;
   Flow_Change_Step : INT;
   Flow_Temp : BOOL;   // 1 - Flow Control/ 0 - Temp Control
   FVIR_1_S_Step : INT;
   FVIR_1_W_Step : INT;
   FVIR_2_S_Step : INT;
   FVIR_2_W_Step : INT;
   FVIR_3_S_Step : INT;
   FVIR_3_W_Step : INT;
   FVIR_4_S_Step : INT;
   FVIR_4_W_Step : INT;
   FVIR_Gas_Flow_Heater_Indication_1 : BOOL;
   FVIR_Gas_Flow_Heater_Indication_2 : BOOL;
   FVIR_Gas_Mass_Flow_FI0011 : REAL := 4.2;
   FVIR_Gas_Mass_Flow_FI0012 : REAL := 10.5;
   FVIR_Gas_SCPM_FI001 : REAL := 0.1483208;
   FVIR_Gas_SCPM_FI0012 : REAL := 0.370802;
   FVIR_LabView_Comm_OK : BOOL;
   FVIR_Water_DRK375 : REAL := 50.0;
   FVIR_Water_DRK375_Error : REAL := -730.0;
   FVIR_Water_float : REAL := 18.0;
   FVIR_Water_Flow_DRK375_REG : REAL := -730.0;
   FVIR_Water_Flow_DRK375_SP : INT;
   FVIR_Water_Outler_Flow : REAL;
   FVIR_Water_Outlet : PID := (CTL := 33555328, CA := 1, DVPA := 1, PVLA := 1, PVHA := 1, KP := 1.0, KI := 0.1, MAXS := 4095.0, MAXO := 50.0, MINO := 25.0, UPD := 0.1, ERR := 50.0, PVH := 200.0, DVP := 100.0, MAXI := 4095.0, MAXTIE := 4095.0, DATA[3] := 50.0, DATA[4] := 50.0, DATA[5] := 0.024420025, DATA[6] := 1.0, DATA[7] := 0.8, DATA[16] := 0.024420025);
   FVIR_Water_Outlet_2 : PID := (CTL := 8422528, PE := 1, INI := 1, DVNA := 1, PVHA := 1, SP := 3.0, KP := 1.0, KI := 0.1, MAXS := 4095.0, SO := 65.760735, MAXO := 100.0, UPD := 0.1, PV := 3.01, ERR := -0.00999999, OUT := 65.760735, MAXI := 4095.0, MAXTIE := 4095.0, DATA[0] := 65.76098, DATA[1] := -1.1760684, DATA[2] := 3.01, DATA[3] := -0.00999999, DATA[4] := 3.0, DATA[5] := 0.024420025, DATA[6] := 1.0, DATA[7] := 1.6, DATA[8] := 1.0, DATA[9] := 0.1, DATA[11] := 1.0, DATA[12] := 0.16666667, DATA[16] := 0.024420025);
   FVIR_Water_Outlet_Valve_Flow_SP_old : REAL;
   FVIR_Water_Outlet_Valve_PID : REAL;
   FVIR_Water_Outlet_Valve_SP_old : REAL;
   FVIR_Water_SP_float : REAL := 20.42;
   FVIR_Water_Temp_DRK375_SP : INT;
   FVIR_Water_Temp_float : REAL := 6.552;
   FVIR_Water_Temp_SP_float : REAL := 7.552;
   Gasoline_Step : SINT;
   GasSolenoidOnOff : BOOL := 1;
   LabView_Stat_B0 : SINT;
   LabView_Stat_B1 : SINT;
   LabView_Stat_B2B3 : DINT;
   LDO_DRK375_Start : BOOL;
   Mannequin_Direction_TimeDelay : INT := 1000;
   Mannequin_GoTo_Home : BOOL;
   Mannequin_GoTo_Work : BOOL;
   Mannequin_Step : DINT;
   Mannequin_Time_Pause : INT := 60;
   Manual : Output_FVIR;
   Modbus_Status_Temp : DINT;
   Number_Mannequin_Movement : INT := 3;
   puls_start : BOOL;
   puls_stop : BOOL;
   Pulse : BOOL[32];
   Reserve : INT;
   Spill_Gasoline_Ons : BOOL;
   Spill_GoTo_Home : BOOL;
   Spill_GoTo_Work : BOOL;
   Start_Manequinn_Move : BOOL;
   Start_Manequinn_Seq : BOOL;
   Start_Manequinn_Seq_Man : BOOL;
   Start_Spill_Gasoline : BOOL;
   Start_Water_Flow : BOOL;
   Start_Water_Flow_T1S : BOOL;
   Start_Water_Flow_T1W : BOOL;
   Start_Water_Flow_T2S : BOOL;
   Start_Water_Flow_T2W : BOOL;
   Start_Water_Flow_T3S : BOOL;
   Start_Water_Flow_T3W : BOOL;
   Start_Water_Flow_T4S : BOOL;
   Start_Water_Flow_T4W : BOOL;
   Temp_Change_Step : INT;
   Temp_Var : INT;
   test : BOOL;
   Tigger_First_Manniquine_Seq : BOOL;
   Timer_Delay : TIMER[30] := ([0].PRE := 250, [1].PRE := 200, [2].PRE := 500, [3].PRE := 500, [4].PRE := 60000, [5].PRE := 1300, [6].PRE := 1300, [7].PRE := 60000, [8].PRE := 10, [9].PRE := 60000, [10].PRE := 3000, [11].PRE := 10, [12].PRE := 60000, [13].PRE := 60000, [14].PRE := 3300000, [15].PRE := 300000, [16].PRE := 3300000, [20].PRE := 60000, [21].PRE := 60000, [25].PRE := 2000, [26].PRE := 2000, [26].ACC := 2000, [27].PRE := 2000, [28].PRE := 2000, [28].ACC := 2000);
   tof0_1sPulse : TIMER := (PRE := 100, ACC := 100);
   tof10sPulse : TIMER := (PRE := 10000, ACC := 8205, TT := 1, DN := 1);
   tof1sPulse : TIMER := (PRE := 500, ACC := 500);
   tof2sPulse : TIMER := (PRE := 2000, ACC := 197, TT := 1, DN := 1);
   ton0 : TIMER;
   ton0_1sPulse : TIMER := (PRE := 100);
   ton10sPulse : TIMER := (PRE := 10000);
   ton1sPulse : TIMER := (PRE := 500, ACC := 205, EN := 1, TT := 1);
   ton2sPulse : TIMER := (PRE := 2000);
   TON_LifeBit_OFF : TIMER := (PRE := 10000);
   TON_LifeBit_ON : TIMER := (PRE := 10000, ACC := 10000, EN := 1, DN := 1);
   Water_Flow_Calc : REAL := 3613.7852;
   Water_Flow_Calc_float : REAL := 8363.267;
   Water_Flow_DRK375 : INT := 8363;
   Water_Flow_DRK375_Last : REAL := 100.0;
   Water_Outlet_Calc : REAL;
   Water_Outlet_Flow_OK : BOOL;
   Water_Outlet_InRange : BOOL := 1;
   Water_Outlet_Valve : INT := 55;
   Water_Temp_Calc : REAL := 2107.655;
   Water_Temp_Calc_float : REAL := 3093.016;
   Water_Temp_DRK375 : INT := 3093;
   Water_Temp_DRK375_Last : REAL := 70.0;
END_VAR

ROUTINE FVIR_Analog_Input   (* ladder *)
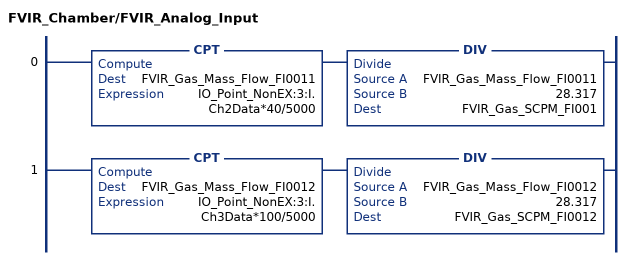
   0: CPT(FVIR_Gas_Mass_Flow_FI0011,IO_Point_NonEX:3:I.Ch2Data*40/5000)DIV(FVIR_Gas_Mass_Flow_FI0011,28.317,FVIR_Gas_SCPM_FI001);
   1: CPT(FVIR_Gas_Mass_Flow_FI0012,IO_Point_NonEX:3:I.Ch3Data*100/5000)DIV(FVIR_Gas_Mass_Flow_FI0012,28.317,FVIR_Gas_SCPM_FI0012);
END_ROUTINE

ROUTINE FVIR_Control_Valve   (* ladder *)
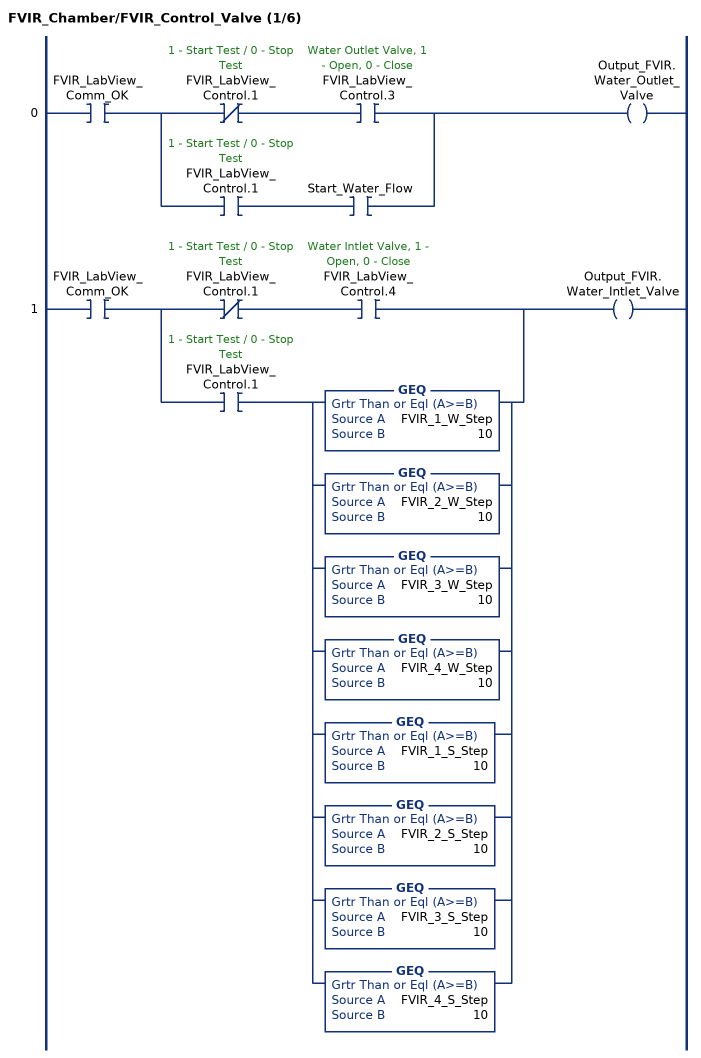
   0: XIC(FVIR_LabView_Comm_OK)[XIO(FVIR_LabView_Control.1) XIC(FVIR_LabView_Control.3) ,XIC(FVIR_LabView_Control.1) XIC(Start_Water_Flow) ]OTE(Output_FVIR.Water_Outlet_Valve);
   1: XIC(FVIR_LabView_Comm_OK)[XIO(FVIR_LabView_Control.1) XIC(FVIR_LabView_Control.4) ,XIC(FVIR_LabView_Control.1) [GEQ(FVIR_1_W_Step,10) ,GEQ(FVIR_2_W_Step,10) ,GEQ(FVIR_3_W_Step,10) ,GEQ(FVIR_4_W_Step,10) ,GEQ(FVIR_1_S_Step,10) ,GEQ(FVIR_2_S_Step,10) ,GEQ(FVIR_3_S_Step,10) ,GEQ(FVIR_4_S_Step,10) ] ]OTE(Output_FVIR.Water_Intlet_Valve);
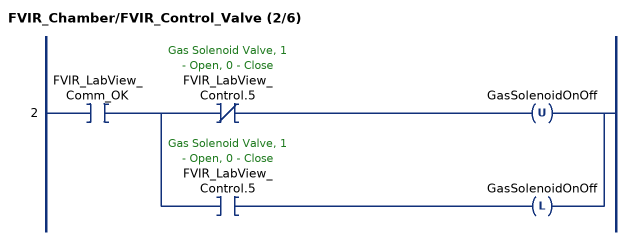
   2: XIC(FVIR_LabView_Comm_OK)[XIO(FVIR_LabView_Control.5) OTU(GasSolenoidOnOff) ,XIC(FVIR_LabView_Control.5) OTL(GasSolenoidOnOff) ];
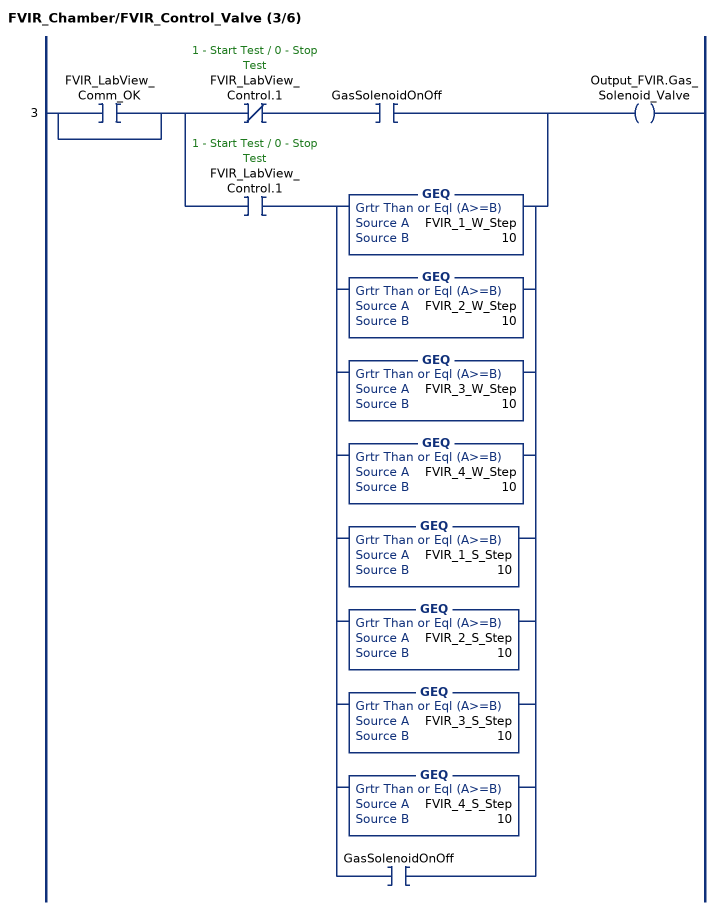
   3: [XIC(FVIR_LabView_Comm_OK) ,][XIO(FVIR_LabView_Control.1) XIC(GasSolenoidOnOff) ,XIC(FVIR_LabView_Control.1) [GEQ(FVIR_1_W_Step,10) ,GEQ(FVIR_2_W_Step,10) ,GEQ(FVIR_3_W_Step,10) ,GEQ(FVIR_4_W_Step,10) ,GEQ(FVIR_1_S_Step,10) ,GEQ(FVIR_2_S_Step,10) ,GEQ(FVIR_3_S_Step,10) ,GEQ(FVIR_4_S_Step,10) ,XIC(GasSolenoidOnOff) ] ]OTE(Output_FVIR.Gas_Solenoid_Valve);
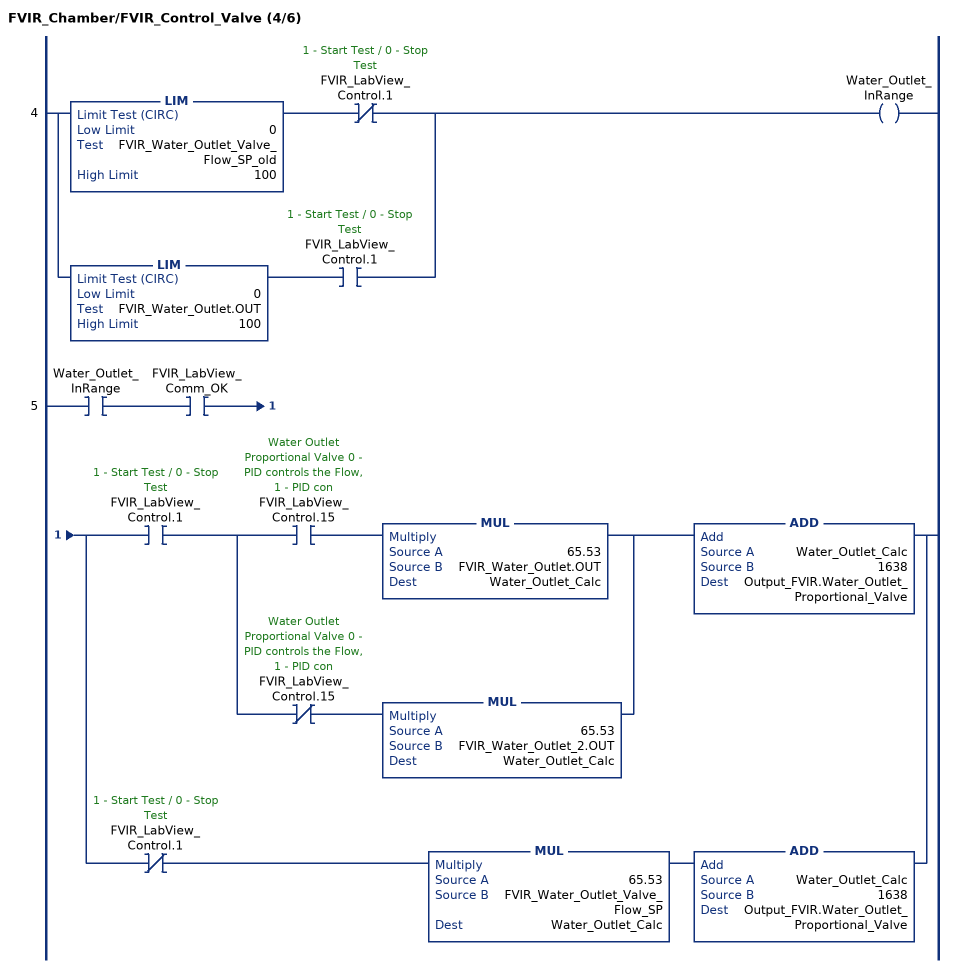
   4: [LIM(0,FVIR_Water_Outlet_Valve_Flow_SP_old,100) XIO(FVIR_LabView_Control.1) ,LIM(0,FVIR_Water_Outlet.OUT,100) XIC(FVIR_LabView_Control.1) ]OTE(Water_Outlet_InRange);
   5: XIC(Water_Outlet_InRange)XIC(FVIR_LabView_Comm_OK)[XIC(FVIR_LabView_Control.1) [XIC(FVIR_LabView_Control.15) MUL(65.53,FVIR_Water_Outlet.OUT,Water_Outlet_Calc) ,XIO(FVIR_LabView_Control.15) MUL(65.53,FVIR_Water_Outlet_2.OUT,Water_Outlet_Calc) ] ADD(Water_Outlet_Calc,1638,Output_FVIR.Water_Outlet_Proportional_Valve) ,XIO(FVIR_LabView_Control.1) MUL(65.53,FVIR_Water_Outlet_Valve_Flow_SP,Water_Outlet_Calc) ADD(Water_Outlet_Calc,1638,Output_FVIR.Water_Outlet_Proportional_Valve) ];
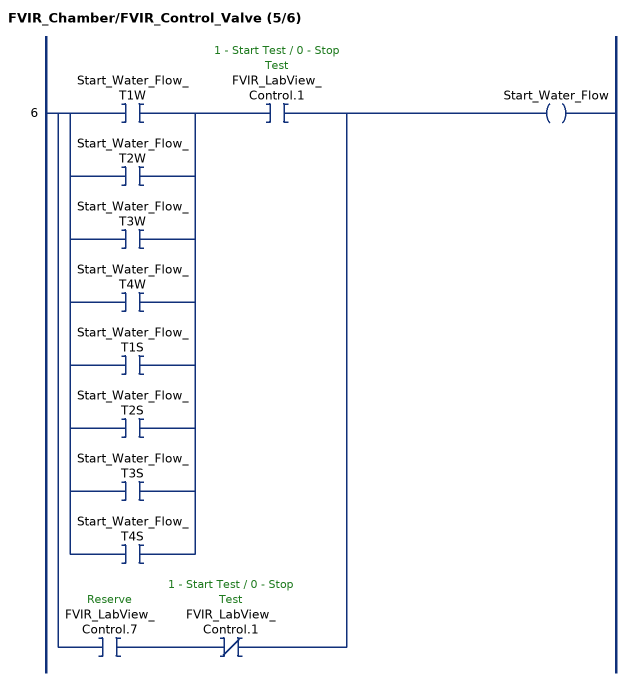
   6: [[XIC(Start_Water_Flow_T1W) ,XIC(Start_Water_Flow_T2W) ,XIC(Start_Water_Flow_T3W) ,XIC(Start_Water_Flow_T4W) ,XIC(Start_Water_Flow_T1S) ,XIC(Start_Water_Flow_T2S) ,XIC(Start_Water_Flow_T3S) ,XIC(Start_Water_Flow_T4S) ] XIC(FVIR_LabView_Control.1) ,XIC(FVIR_LabView_Control.7) XIO(FVIR_LabView_Control.1) ]OTE(Start_Water_Flow);
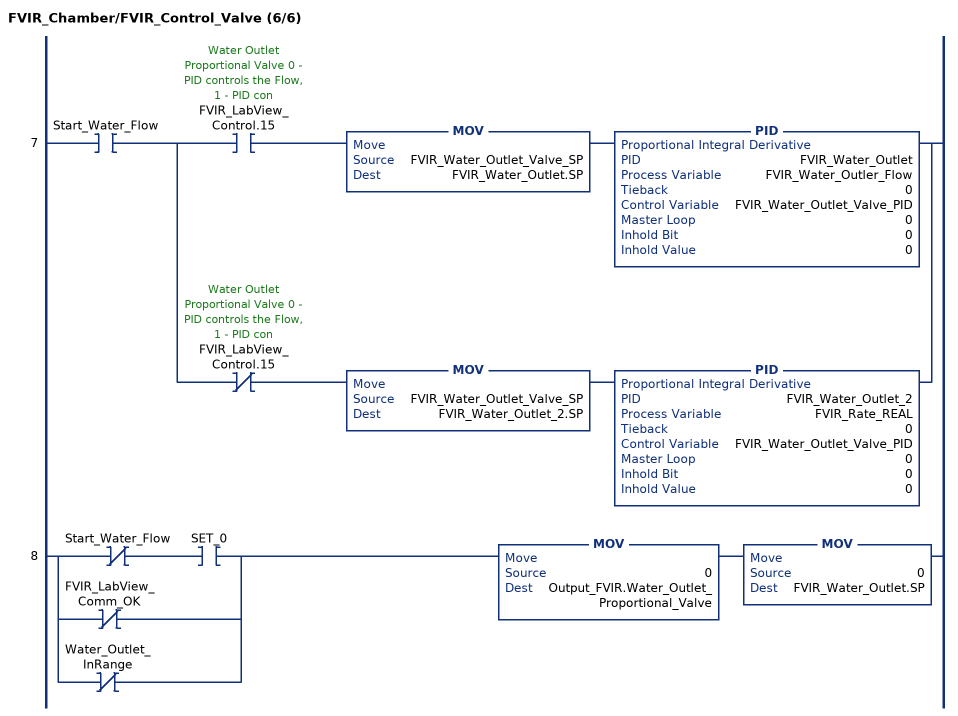
   7: XIC(Start_Water_Flow)[XIC(FVIR_LabView_Control.15) MOV(FVIR_Water_Outlet_Valve_SP,FVIR_Water_Outlet.SP) PID(FVIR_Water_Outlet,FVIR_Water_Outler_Flow,0,FVIR_Water_Outlet_Valve_PID,0,0,0) ,XIO(FVIR_LabView_Control.15) MOV(FVIR_Water_Outlet_Valve_SP,FVIR_Water_Outlet_2.SP) PID(FVIR_Water_Outlet_2,FVIR_Rate_REAL,0,FVIR_Water_Outlet_Valve_PID,0,0,0) ];
   8: [XIO(Start_Water_Flow) XIC(SET_0) ,XIO(FVIR_LabView_Comm_OK) ,XIO(Water_Outlet_InRange) ]MOV(0,Output_FVIR.Water_Outlet_Proportional_Valve)MOV(0,FVIR_Water_Outlet.SP);
END_ROUTINE

ROUTINE FVIR_Error_MSG   (* ladder *)
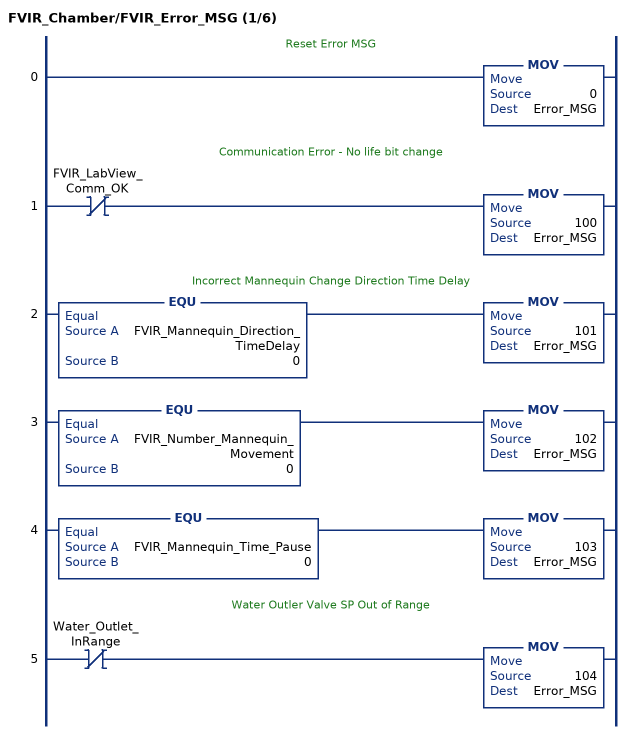
   // Reset Error MSG
   0: MOV(0,Error_MSG);
   // Communication Error - No life bit change
   1: XIO(FVIR_LabView_Comm_OK)MOV(100,Error_MSG);
   // Incorrect Mannequin Change Direction Time Delay
   2: EQU(FVIR_Mannequin_Direction_TimeDelay,0)MOV(101,Error_MSG);
   3: EQU(FVIR_Number_Mannequin_Movement,0)MOV(102,Error_MSG);
   4: EQU(FVIR_Mannequin_Time_Pause,0)MOV(103,Error_MSG);
   // Water Outler Valve SP Out of Range
   5: XIO(Water_Outlet_InRange)MOV(104,Error_MSG);
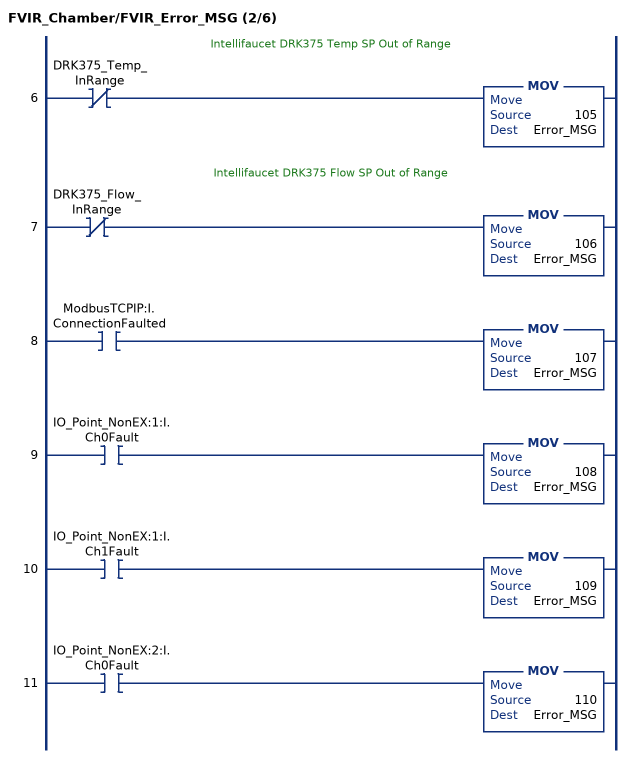
   // Intellifaucet DRK375 Temp SP Out of Range
   6: XIO(DRK375_Temp_InRange)MOV(105,Error_MSG);
   // Intellifaucet DRK375 Flow SP Out of Range
   7: XIO(DRK375_Flow_InRange)MOV(106,Error_MSG);
   8: XIC(ModbusTCPIP:I.ConnectionFaulted)MOV(107,Error_MSG);
   9: XIC(IO_Point_NonEX:1:I.Ch0Fault)MOV(108,Error_MSG);
   10: XIC(IO_Point_NonEX:1:I.Ch1Fault)MOV(109,Error_MSG);
   11: XIC(IO_Point_NonEX:2:I.Ch0Fault)MOV(110,Error_MSG);
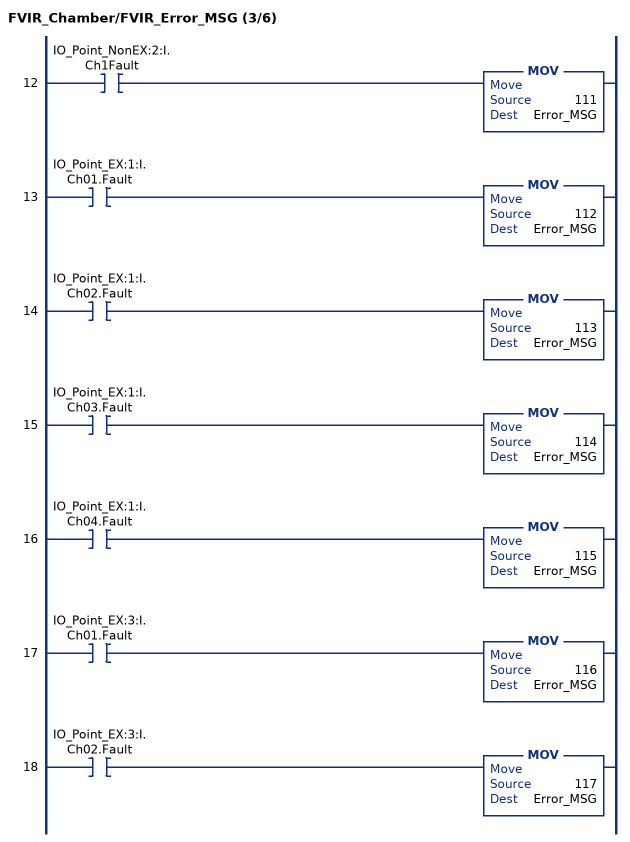
   12: XIC(IO_Point_NonEX:2:I.Ch1Fault)MOV(111,Error_MSG);
   13: XIC(IO_Point_EX:1:I.Ch01.Fault)MOV(112,Error_MSG);
   14: XIC(IO_Point_EX:1:I.Ch02.Fault)MOV(113,Error_MSG);
   15: XIC(IO_Point_EX:1:I.Ch03.Fault)MOV(114,Error_MSG);
   16: XIC(IO_Point_EX:1:I.Ch04.Fault)MOV(115,Error_MSG);
   17: XIC(IO_Point_EX:3:I.Ch01.Fault)MOV(116,Error_MSG);
   18: XIC(IO_Point_EX:3:I.Ch02.Fault)MOV(117,Error_MSG);
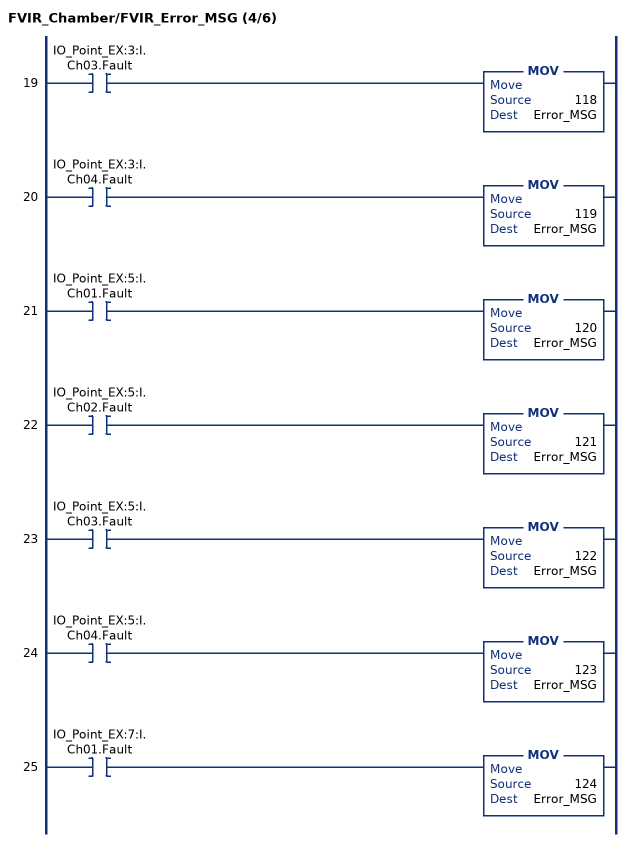
   19: XIC(IO_Point_EX:3:I.Ch03.Fault)MOV(118,Error_MSG);
   20: XIC(IO_Point_EX:3:I.Ch04.Fault)MOV(119,Error_MSG);
   21: XIC(IO_Point_EX:5:I.Ch01.Fault)MOV(120,Error_MSG);
   22: XIC(IO_Point_EX:5:I.Ch02.Fault)MOV(121,Error_MSG);
   23: XIC(IO_Point_EX:5:I.Ch03.Fault)MOV(122,Error_MSG);
   24: XIC(IO_Point_EX:5:I.Ch04.Fault)MOV(123,Error_MSG);
   25: XIC(IO_Point_EX:7:I.Ch01.Fault)MOV(124,Error_MSG);
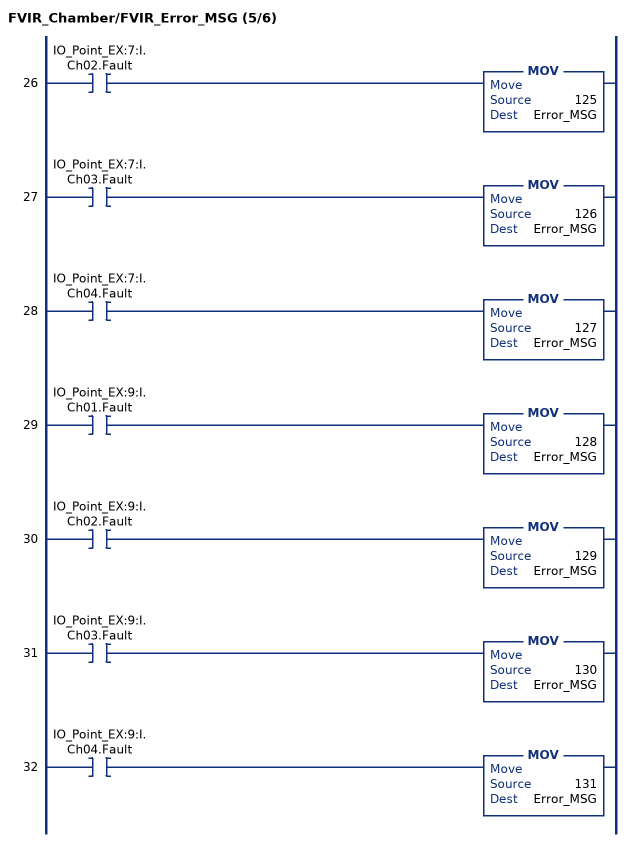
   26: XIC(IO_Point_EX:7:I.Ch02.Fault)MOV(125,Error_MSG);
   27: XIC(IO_Point_EX:7:I.Ch03.Fault)MOV(126,Error_MSG);
   28: XIC(IO_Point_EX:7:I.Ch04.Fault)MOV(127,Error_MSG);
   29: XIC(IO_Point_EX:9:I.Ch01.Fault)MOV(128,Error_MSG);
   30: XIC(IO_Point_EX:9:I.Ch02.Fault)MOV(129,Error_MSG);
   31: XIC(IO_Point_EX:9:I.Ch03.Fault)MOV(130,Error_MSG);
   32: XIC(IO_Point_EX:9:I.Ch04.Fault)MOV(131,Error_MSG);
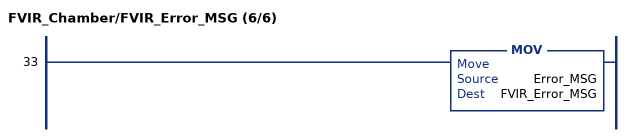
   33: MOV(Error_MSG,FVIR_Error_MSG);
END_ROUTINE

ROUTINE FVIR_Intellfaucet_Control   (* ladder *)
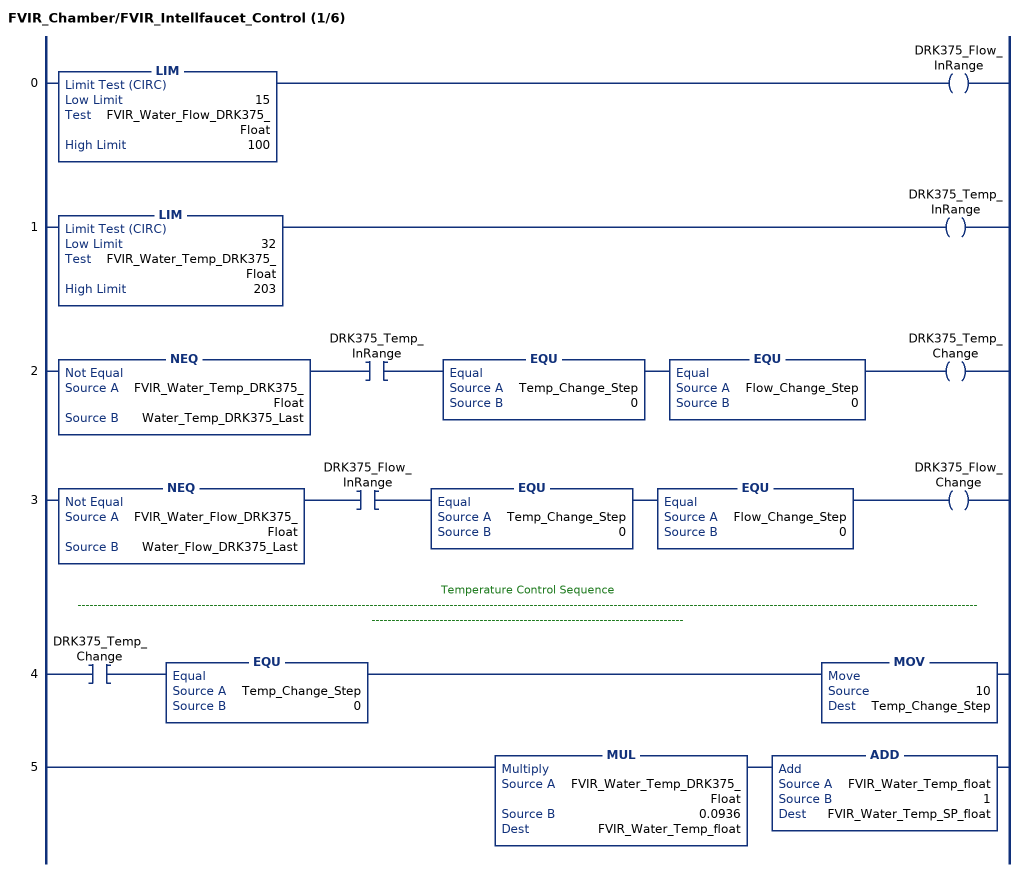
   0: LIM(15,FVIR_Water_Flow_DRK375_Float,100)OTE(DRK375_Flow_InRange);
   1: LIM(32,FVIR_Water_Temp_DRK375_Float,203)OTE(DRK375_Temp_InRange);
   2: NEQ(FVIR_Water_Temp_DRK375_Float,Water_Temp_DRK375_Last)XIC(DRK375_Temp_InRange)EQU(Temp_Change_Step,0)EQU(Flow_Change_Step,0)OTE(DRK375_Temp_Change);
   3: NEQ(FVIR_Water_Flow_DRK375_Float,Water_Flow_DRK375_Last)XIC(DRK375_Flow_InRange)EQU(Temp_Change_Step,0)EQU(Flow_Change_Step,0)OTE(DRK375_Flow_Change);
   // Temperature Control Sequence
   // ---------------------------------------------------------------------------------------------------------------------------------------------------------------------------------------------------------------------------------------------------------------------------------------------------------------
   4: XIC(DRK375_Temp_Change)EQU(Temp_Change_Step,0)MOV(10,Temp_Change_Step);
   5: MUL(FVIR_Water_Temp_DRK375_Float,0.0936,FVIR_Water_Temp_float)ADD(FVIR_Water_Temp_float,1,FVIR_Water_Temp_SP_float);
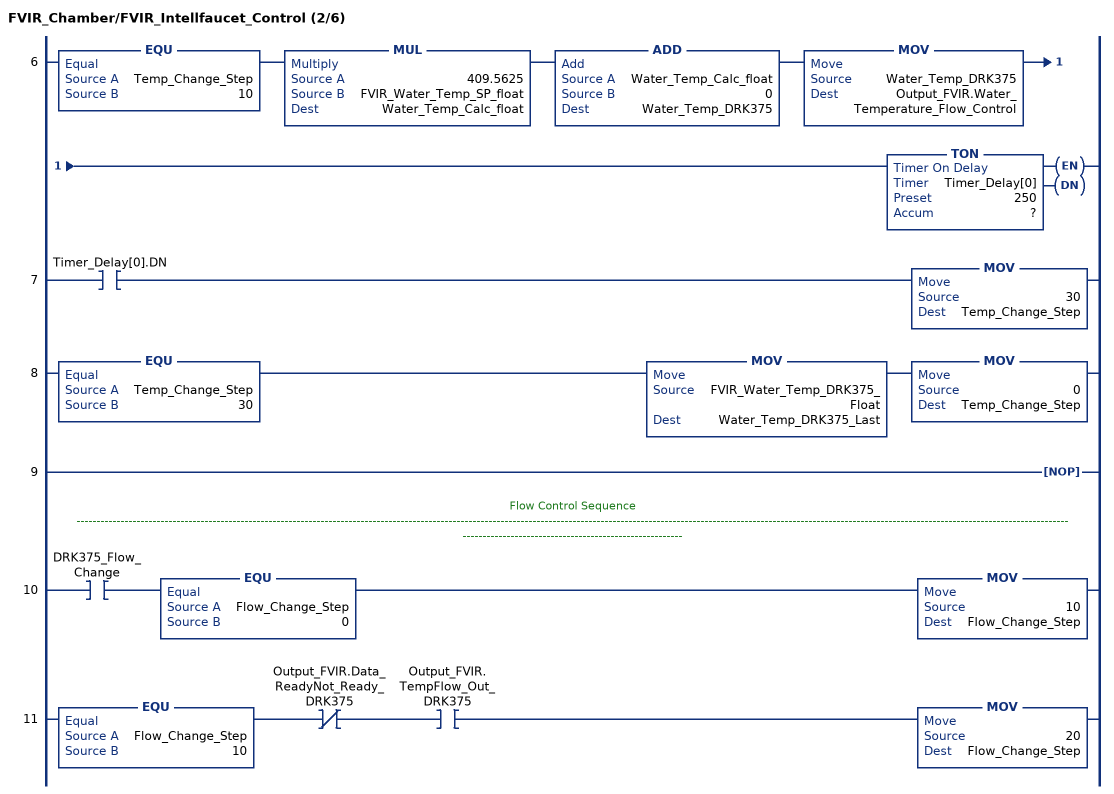
   6: EQU(Temp_Change_Step,10)MUL(409.5625,FVIR_Water_Temp_SP_float,Water_Temp_Calc_float)ADD(Water_Temp_Calc_float,0,Water_Temp_DRK375)MOV(Water_Temp_DRK375,Output_FVIR.Water_Temperature_Flow_Control)TON(Timer_Delay[0],?,?);
   7: XIC(Timer_Delay[0].DN)MOV(30,Temp_Change_Step);
   8: EQU(Temp_Change_Step,30)MOV(FVIR_Water_Temp_DRK375_Float,Water_Temp_DRK375_Last)MOV(0,Temp_Change_Step);
   9: NOP();
   // Flow Control Sequence
   // ---------------------------------------------------------------------------------------------------------------------------------------------------------------------------------------------------------------------------------------------------------------------------------------------------------------
   10: XIC(DRK375_Flow_Change)EQU(Flow_Change_Step,0)MOV(10,Flow_Change_Step);
   11: EQU(Flow_Change_Step,10)XIO(Output_FVIR.Data_ReadyNot_Ready_DRK375)XIC(Output_FVIR.TempFlow_Out_DRK375)MOV(20,Flow_Change_Step);
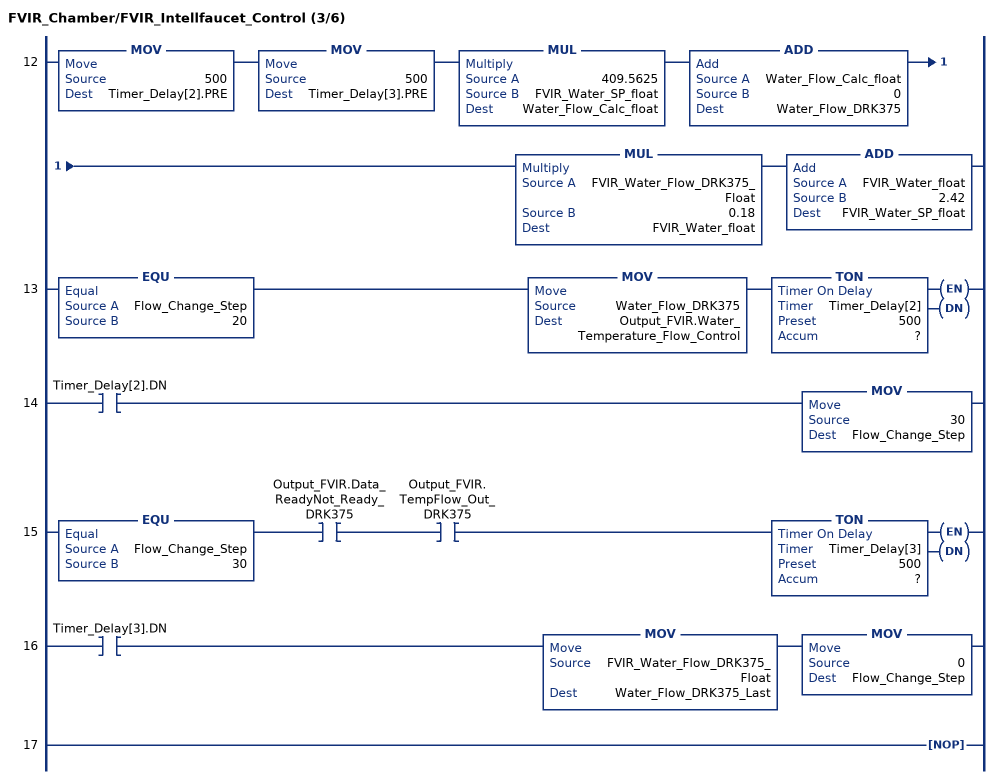
   12: MOV(500,Timer_Delay[2].PRE)MOV(500,Timer_Delay[3].PRE)MUL(409.5625,FVIR_Water_SP_float,Water_Flow_Calc_float)ADD(Water_Flow_Calc_float,0,Water_Flow_DRK375)MUL(FVIR_Water_Flow_DRK375_Float,0.18,FVIR_Water_float)ADD(FVIR_Water_float,2.42,FVIR_Water_SP_float);
   13: EQU(Flow_Change_Step,20)MOV(Water_Flow_DRK375,Output_FVIR.Water_Temperature_Flow_Control)TON(Timer_Delay[2],?,?);
   14: XIC(Timer_Delay[2].DN)MOV(30,Flow_Change_Step);
   15: EQU(Flow_Change_Step,30)XIC(Output_FVIR.Data_ReadyNot_Ready_DRK375)XIC(Output_FVIR.TempFlow_Out_DRK375)TON(Timer_Delay[3],?,?);
   16: XIC(Timer_Delay[3].DN)MOV(FVIR_Water_Flow_DRK375_Float,Water_Flow_DRK375_Last)MOV(0,Flow_Change_Step);
   17: NOP();
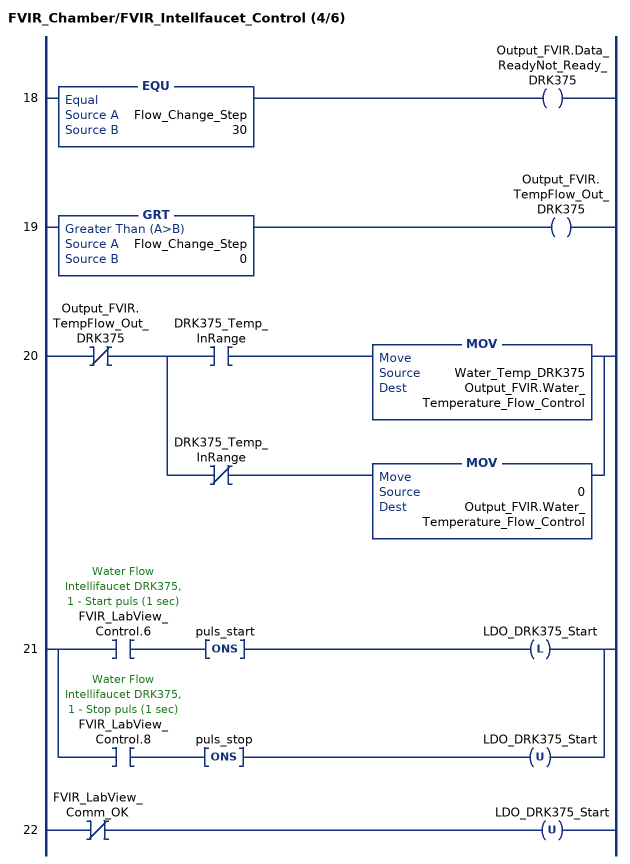
   18: EQU(Flow_Change_Step,30)OTE(Output_FVIR.Data_ReadyNot_Ready_DRK375);
   19: GRT(Flow_Change_Step,0)OTE(Output_FVIR.TempFlow_Out_DRK375);
   20: XIO(Output_FVIR.TempFlow_Out_DRK375)[XIC(DRK375_Temp_InRange) MOV(Water_Temp_DRK375,Output_FVIR.Water_Temperature_Flow_Control) ,XIO(DRK375_Temp_InRange) MOV(0,Output_FVIR.Water_Temperature_Flow_Control) ];
   21: [XIC(FVIR_LabView_Control.6) ONS(puls_start) OTL(LDO_DRK375_Start) ,XIC(FVIR_LabView_Control.8) ONS(puls_stop) OTU(LDO_DRK375_Start) ];
   22: XIO(FVIR_LabView_Comm_OK)OTU(LDO_DRK375_Start);
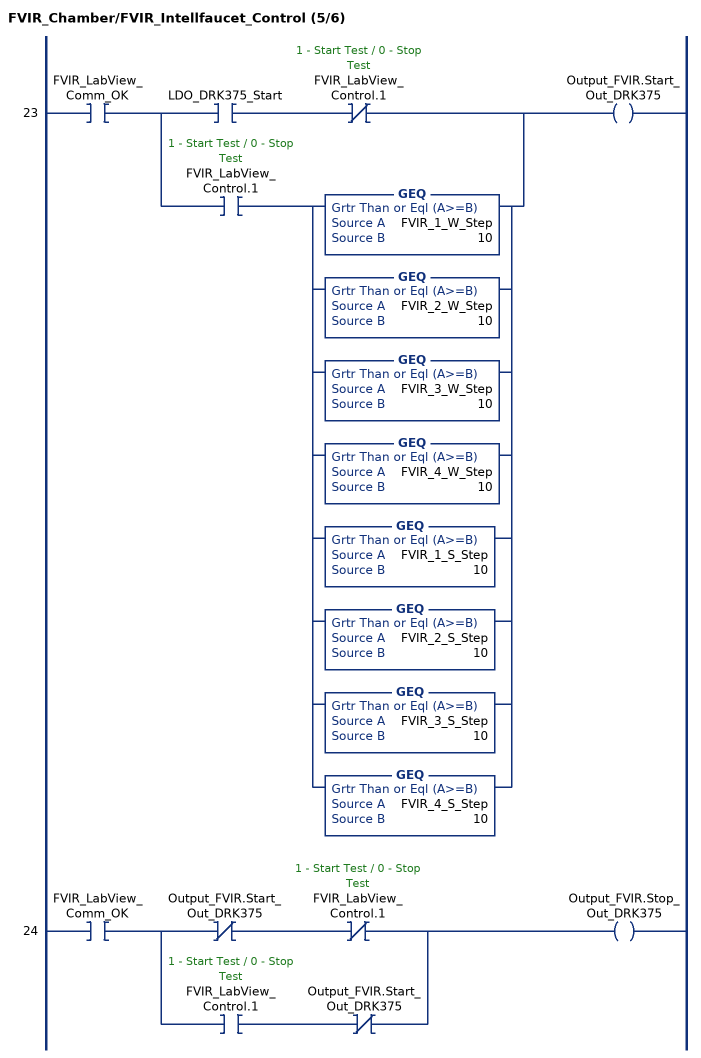
   23: XIC(FVIR_LabView_Comm_OK)[XIC(LDO_DRK375_Start) XIO(FVIR_LabView_Control.1) ,XIC(FVIR_LabView_Control.1) [GEQ(FVIR_1_W_Step,10) ,GEQ(FVIR_2_W_Step,10) ,GEQ(FVIR_3_W_Step,10) ,GEQ(FVIR_4_W_Step,10) ,GEQ(FVIR_1_S_Step,10) ,GEQ(FVIR_2_S_Step,10) ,GEQ(FVIR_3_S_Step,10) ,GEQ(FVIR_4_S_Step,10) ] ]OTE(Output_FVIR.Start_Out_DRK375);
   24: XIC(FVIR_LabView_Comm_OK)[XIO(Output_FVIR.Start_Out_DRK375) XIO(FVIR_LabView_Control.1) ,XIC(FVIR_LabView_Control.1) XIO(Output_FVIR.Start_Out_DRK375) ]OTE(Output_FVIR.Stop_Out_DRK375);
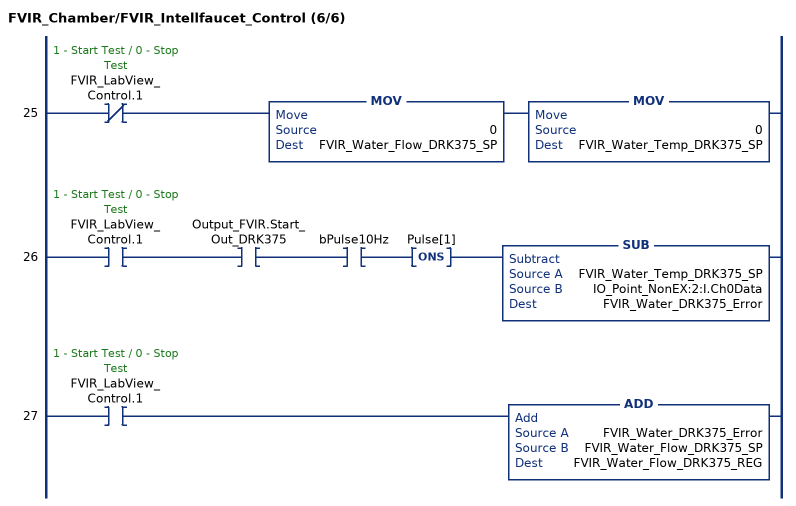
   25: XIO(FVIR_LabView_Control.1)MOV(0,FVIR_Water_Flow_DRK375_SP)MOV(0,FVIR_Water_Temp_DRK375_SP);
   26: XIC(FVIR_LabView_Control.1)XIC(Output_FVIR.Start_Out_DRK375)XIC(bPulse10Hz)ONS(Pulse[1])SUB(FVIR_Water_Temp_DRK375_SP,IO_Point_NonEX:2:I.Ch0Data,FVIR_Water_DRK375_Error);
   27: XIC(FVIR_LabView_Control.1)ADD(FVIR_Water_DRK375_Error,FVIR_Water_Flow_DRK375_SP,FVIR_Water_Flow_DRK375_REG);
END_ROUTINE
